(* CoDeSys 2.3 export: CHECKDIVWORD.EXP *)

(* POU CheckDivWord, ST *)
FUNCTION CheckDivWord : WORD
VAR_INPUT
	divisor: WORD;
END_VAR
VAR
END_VAR
(* @TEXT_IMPLEMENTATION := 'ST' *)
IF divisor = 0 THEN
	CheckDivWord := 1;
ELSE
	CheckDivWord := divisor;
END_IF
END_FUNCTION
